PROGRAM pouS6Warnings
VAR
	
idbMsgWarn: FB_CheckMessageBounds;
END_VAR

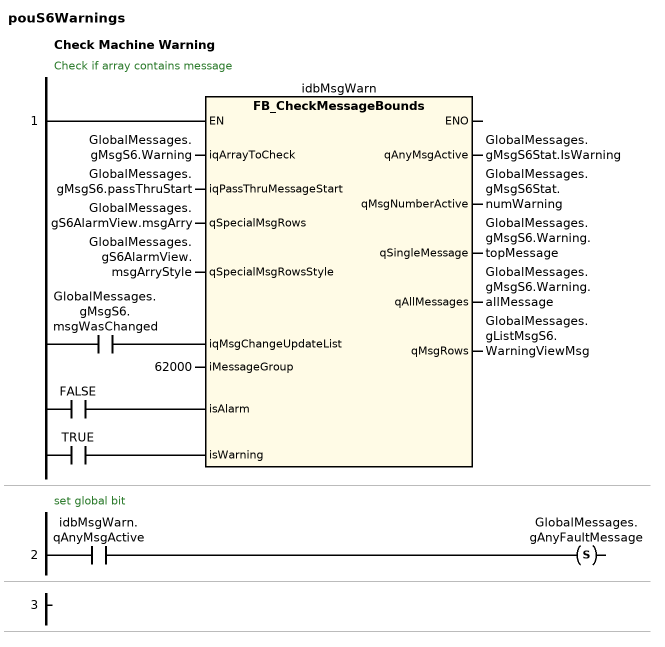
// NETWORK 1: Check Machine Warning
// Check if array contains message
idbMsgWarn(
    iqArrayToCheck := GlobalMessages.gMsgS6.Warning,
    iqPassThruMessageStart := GlobalMessages.gMsgS6.passThruStart,
    qSpecialMsgRows := GlobalMessages.gS6AlarmView.msgArry,
    qSpecialMsgRowsStyle := GlobalMessages.gS6AlarmView.msgArryStyle,
    iqMsgChangeUpdateList := GlobalMessages.gMsgS6.msgWasChanged,
    iMessageGroup := 62000,
    isAlarm := FALSE,
    isWarning := TRUE,
    qAnyMsgActive => GlobalMessages.gMsgS6Stat.IsWarning,
    qMsgNumberActive => GlobalMessages.gMsgS6Stat.numWarning,
    qSingleMessage => GlobalMessages.gMsgS6.Warning.topMessage,
    qAllMessages => GlobalMessages.gMsgS6.Warning.allMessage,
    qMsgRows => GlobalMessages.gListMsgS6.WarningViewMsg); // FB_CheckMessageBounds

// NETWORK 2
// set global bit
GlobalMessages.gAnyFaultMessage S= idbMsgWarn.qAnyMsgActive;

// NETWORK 3

END_PROGRAM

(* stored: Version 1.1.0.1, ProductVersion 3.1.4024.12
   POU pouS6Warnings: Id {b3787da7-6c25-4881-be08-a57d4d9bdeab}, SpecialFunc None *)
